Yaskawa INFORM job: driller_case_upwards_planes_program.JBI

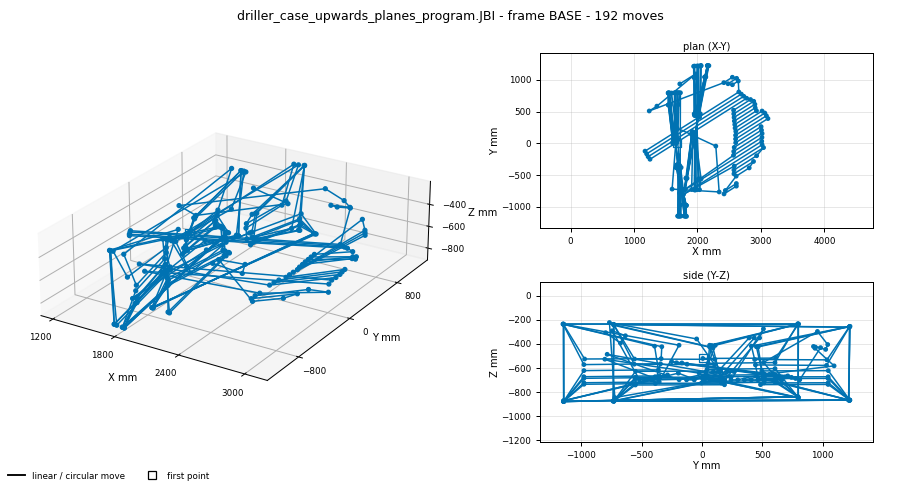
[picture p0: tool path of driller_case_upwards_planes_program.JBI in frame BASE, 192 of 196 moves have a stored position in this frame; points joined in program order, loops and branches not executed]
/JOB
//NAME driller_case_upwards_planes_program
//POS
///NPOS 192,0,192,0,0,0
///TOOL 0
///POSTYPE BASE
///RECTAN
///RCONF 0,0,0,0,0,0,0,0,0,0,0,0,0,0,0,0,0,0,0,0,0,0,0,0
C00000=1673.431880,7.470572,-520.659280,175.000000,-87.408482,-5.000000
C00001=1701.430434,612.195440,-517.792634,5.000000,-89.787348,-140.532242
C00002=1730.822135,797.239311,-237.810218,175.000000,-61.554488,-43.406673
C00003=1724.400104,-1148.148230,-235.635493,175.000000,-56.840650,28.530040
C00004=1729.963488,-971.443104,-525.203951,175.000000,-89.826502,-50.531598
C00005=1674.986268,-337.641847,-522.278767,168.678223,-90.000000,5.000000
C00006=1704.945690,-332.291816,-423.533285,5.000000,-42.547616,175.000000
C00007=1691.135780,-1145.204123,-238.489082,175.000000,-58.717311,26.416525
C00008=1739.409858,-1145.531949,-872.838304,-5.000000,-56.170316,-151.289669
C00009=1742.002509,-379.860852,-686.285449,175.000000,-48.174345,-17.109685
C00010=1678.244549,-343.199867,-564.964424,168.678223,-90.000000,5.000000
C00011=1818.384608,-977.621480,-571.536946,-175.000000,-89.631981,-46.846842
C00012=1826.808543,-1150.833072,-235.822537,175.000000,-54.888634,30.707899
C00013=1590.979545,793.251519,-233.985937,-175.000000,-62.535779,-40.616460
C00014=1571.245197,605.149655,-554.917240,5.000000,-89.484561,-136.850153
C00015=1625.513935,50.641867,-560.809912,168.678223,-90.000000,5.000000
C00016=1689.473871,63.888821,-411.282587,-5.000000,-48.045317,175.000000
C00017=1708.256775,799.356476,-235.389466,175.000000,-61.004563,-44.985899
C00018=1636.215691,796.253953,-843.502997,-5.000000,-63.369743,139.463298
C00019=1641.861992,13.097528,-670.904228,175.000000,-43.584726,-21.662339
C00020=1619.863907,43.091049,-610.639771,168.678223,-90.000000,5.000000
C00021=1564.744394,605.389718,-604.672433,5.000000,-89.485299,-136.858461
C00022=1558.133538,794.132963,-838.862886,5.000000,-63.890650,140.856457
C00023=1793.575292,-1145.031741,-876.264127,5.000000,-55.710812,-151.382699
C00024=1811.384412,-977.382379,-621.271160,175.000000,-89.632395,-46.855158
C00025=1673.763040,-360.368406,-614.890343,168.678223,-90.000000,5.000000
C00026=1713.133832,-392.278475,-418.917620,5.000000,-45.513699,161.896712
C00027=1701.888861,-1146.465321,-236.949035,175.000000,-57.847486,27.323797
C00028=1714.482776,-1144.136050,-870.078236,-5.000000,-56.959520,-152.294224
C00029=1719.658713,-351.013457,-679.536032,175.000000,-45.302626,-5.000000
C00030=1674.759987,-354.429105,-664.960497,168.678223,-90.000000,5.000000
C00031=1823.436094,-977.958927,-671.848021,175.000000,-89.610377,-46.409872
C00032=1809.321792,-1145.234620,-877.559004,5.000000,-55.428903,-151.169659
C00033=1544.248518,793.640543,-837.946269,5.000000,-64.024640,141.178755
C00034=1549.995593,604.768012,-654.123768,5.000000,-89.445413,-136.413643
C00035=1616.889276,32.814080,-660.602958,168.678223,-90.000000,5.000000
C00036=1669.829005,80.581913,-413.436350,5.000000,-46.334068,-175.000000
C00037=1682.622532,797.248951,-235.622802,175.000000,-61.552203,-43.413607
C00038=1656.620159,798.095359,-846.102626,5.000000,-62.596024,138.067586
C00039=1655.982659,0.583805,-677.340283,175.000000,-46.582826,-23.977786
C00040=1614.845882,21.413497,-710.613338,168.678223,-90.000000,5.000000
C00041=1544.922944,604.889358,-703.953307,5.000000,-89.440488,-136.359327
C00042=1541.265869,793.579835,-837.776448,5.000000,-64.040832,141.218191
C00043=1809.966137,-1145.258187,-877.659798,5.000000,-55.394158,-151.143981
C00044=1821.644860,-977.832954,-721.815313,175.000000,-89.607710,-46.355496
C00045=1671.662160,-353.900735,-714.869605,168.678223,-90.000000,5.000000
C00046=1694.918489,-189.479139,-411.049691,5.000000,-48.693566,-162.669170
C00047=1688.735226,-1145.992617,-237.083073,175.000000,-58.161087,26.984028
C00048=1714.386065,-1144.637206,-870.689055,5.000000,-56.663329,-151.932909
C00049=1723.789184,-403.538739,-698.708952,175.000000,-54.643933,-34.099882
C00050=1673.691517,-382.283167,-678.538009,168.678223,-90.000000,5.000000
C00051=1821.794903,-977.808560,-685.265560,175.000000,-89.602307,-46.245060
C00052=1812.732992,-1145.305389,-877.931109,5.000000,-55.323257,-151.091931
C00053=1536.659104,793.456173,-837.497478,-5.000000,-64.073595,141.298327
C00054=1538.402248,604.904947,-667.123556,-5.000000,-89.430451,-136.249014
C00055=1612.340142,12.697218,-673.988201,168.678223,-90.000000,5.000000
C00056=1668.454091,110.569857,-412.045848,5.000000,-46.959807,-174.665225
C00057=1681.902703,797.234172,-235.601339,-175.000000,-61.556609,-43.402511
C00058=1656.233440,798.109144,-846.096344,5.000000,-62.590789,138.057175
C00059=1656.170573,2.028916,-680.034745,-175.000000,-47.980448,-27.377056
C00060=1610.322073,-2.559617,-724.017037,168.678223,-90.000000,5.000000
C00061=1545.419504,606.009907,-717.420022,-5.000000,-89.472373,-136.713354
C00062=1547.396406,793.973294,-838.282370,-5.000000,-63.934611,140.961437
C00063=1792.490907,-1145.099774,-876.404413,5.000000,-55.619211,-151.312650
C00064=1800.788436,-976.746038,-734.385420,175.000000,-89.625178,-46.709903
C00065=1663.430936,-385.311442,-728.138889,180.000000,-60.000000,0.000000
C00066=2418.072893,-797.339000,-307.192250,175.000000,-13.138131,5.000000
C00067=2612.434723,-674.639778,-393.619264,175.000000,-13.138131,5.000000
C00068=2612.338702,-633.486964,-332.637264,175.000000,-13.138131,5.000000
C00069=2439.090274,-742.857448,-291.122264,175.000000,-13.138131,5.000000
C00070=2609.232584,-517.188349,-698.109264,175.000000,-13.138131,5.000000
C00071=2815.107824,-387.220793,-671.983264,175.000000,-13.138131,5.000000
C00072=2882.831238,-285.337748,-656.650264,175.000000,-13.138131,5.000000
C00073=2574.452592,-480.014964,-698.349264,175.000000,-13.138131,5.000000
C00074=2574.249107,-421.013680,-696.275264,175.000000,-13.138131,5.000000
C00075=2931.745166,-195.328994,-642.567264,175.000000,-13.138131,5.000000
C00076=3040.631451,-67.460124,-690.751264,175.000000,-13.138131,5.000000
C00077=2579.605431,-358.502529,-697.708264,175.000000,-13.138131,5.000000
C00078=1780.417411,-803.894423,-526.918264,175.000000,-13.138131,5.000000
C00079=3018.335870,-22.405421,-642.237264,175.000000,-13.138131,5.000000
C00080=3012.500702,33.040622,-630.532264,175.000000,-13.138131,5.000000
C00081=1716.986018,-784.808462,-486.219264,175.000000,-13.138131,5.000000
C00082=2567.445798,-188.789589,-697.222264,175.000000,-13.138131,5.000000
C00083=3015.932444,94.336798,-631.217264,175.000000,-13.138131,5.000000
C00084=3018.491529,155.082073,-626.978264,175.000000,-13.138131,5.000000
C00085=2571.014527,-127.406933,-697.829264,175.000000,-13.138131,5.000000
C00086=2578.759665,-63.387741,-698.559264,175.000000,-13.138131,5.000000
C00087=3008.587342,207.959374,-627.283264,175.000000,-13.138131,5.000000
C00088=3002.687909,263.364847,-628.708264,175.000000,-13.138131,5.000000
C00089=2601.758547,10.261031,-697.750264,175.000000,-13.138131,5.000000
C00090=2600.088796,68.336671,-698.106264,175.000000,-13.138131,5.000000
C00091=3110.624587,390.634237,-350.634264,175.000000,-13.138131,5.000000
C00092=3086.098318,434.280723,-350.923264,175.000000,-13.138131,5.000000
C00093=2600.297118,127.597926,-698.488264,175.000000,-13.138131,5.000000
C00094=2603.303524,188.625591,-697.822264,175.000000,-13.138131,5.000000
C00095=3061.064690,477.606917,-350.373264,175.000000,-13.138131,5.000000
C00096=3017.690039,509.354554,-275.549264,175.000000,-13.138131,5.000000
C00097=2592.388002,240.864444,-698.256264,175.000000,-13.138131,5.000000
C00098=2587.301189,296.782918,-697.884264,175.000000,-13.138131,5.000000
C00099=2929.507142,512.815070,-646.336264,175.000000,-13.138131,5.000000
C00100=2909.851518,559.536359,-652.328264,175.000000,-13.138131,5.000000
C00101=2580.862263,351.847814,-698.019264,175.000000,-13.138131,5.000000
C00102=2576.339464,408.122346,-698.387264,175.000000,-13.138131,5.000000
C00103=2904.740182,615.439352,-696.121264,175.000000,-13.138131,5.000000
C00104=2886.403691,662.993401,-697.340264,175.000000,-13.138131,5.000000
C00105=2571.376107,464.118757,-698.288264,175.000000,-13.138131,5.000000
C00106=2568.806639,521.626413,-697.221264,175.000000,-13.138131,5.000000
C00107=2835.976752,690.288980,-673.466264,175.000000,-13.138131,5.000000
C00108=2774.286445,710.474076,-664.905264,175.000000,-13.138131,5.000000
C00109=1251.445386,-250.884509,-547.070264,175.000000,-13.138131,5.000000
C00110=1222.182922,-210.227949,-556.282264,175.000000,-13.138131,5.000000
C00111=2729.668764,741.436999,-677.026264,175.000000,-13.138131,5.000000
C00112=2690.657399,775.939148,-686.387264,175.000000,-13.138131,5.000000
C00113=1198.557215,-166.012945,-557.802264,175.000000,-13.138131,5.000000
C00114=1173.125310,-122.938180,-568.494264,175.000000,-13.138131,5.000000
C00115=2651.104851,810.099652,-696.529264,175.000000,-13.138131,5.000000
C00116=2643.398138,982.623688,-430.995264,175.000000,-13.138131,5.000000
C00117=2550.399255,923.914164,-421.281264,175.000000,-13.138131,5.000000
C00118=2481.149301,939.326909,-426.588264,175.000000,-13.138131,5.000000
C00119=2616.445002,1024.738110,-445.606264,175.000000,-13.138131,5.000000
C00120=2549.748754,1041.762992,-405.392264,175.000000,-13.138131,5.000000
C00121=2414.820888,956.584003,-297.084264,175.000000,-13.138131,5.000000
C00122=1239.226227,510.088279,-553.661264,175.000000,-13.138131,5.000000
C00123=1360.051207,586.364219,-645.180264,175.000000,-13.138131,5.000000
C00124=1971.096569,1094.552710,-581.948264,175.000000,-13.138131,5.000000
C00125=1720.950038,936.637008,-436.438264,175.000000,-13.138131,5.000000
C00126=1961.484996,107.194191,-528.136914,5.000000,-87.762077,175.000000
C00127=2016.650761,-558.205833,-525.321042,5.000000,-89.841698,129.060213
C00128=1989.641452,-729.842232,-241.045760,175.000000,-57.590997,26.248990
C00129=1997.453896,1220.092504,-260.476656,-175.000000,-62.729371,-42.375589
C00130=1987.427131,1034.868670,-532.157780,175.000000,-89.803316,39.059669
C00131=1960.156670,436.797064,-529.555779,167.889080,-90.000000,5.000000
C00132=2032.382048,409.596982,-418.437173,-5.000000,-51.077351,163.119403
C00133=2054.997730,1226.570891,-254.753398,175.000000,-61.067124,-47.210966
C00134=1939.009741,1213.927494,-864.805716,5.000000,-64.011021,140.374043
C00135=1947.622597,464.514384,-680.611039,175.000000,-39.536143,-5.000000
C00136=1952.014832,443.273018,-574.460068,167.889080,-90.000000,5.000000
C00137=1948.276945,1032.014046,-578.095382,175.000000,-89.712556,40.386055
C00138=1952.492216,1218.817292,-263.193512,175.000000,-63.172057,-41.437844
C00139=2031.818883,-730.783852,-237.814917,175.000000,-56.842528,26.968983
C00140=2056.236526,-560.610843,-568.391185,5.000000,-89.779417,130.387161
C00141=1969.048653,105.201390,-572.392321,167.889080,-90.000000,5.000000
C00142=2288.843492,-43.671885,-359.161426,5.000000,-71.416390,160.782079
C00143=2341.409332,-766.085094,-223.316094,175.000000,-55.190941,48.507226
C00144=1599.653871,-721.210506,-844.569748,-5.000000,-74.132634,-161.793602
C00145=1676.842950,239.149767,-675.094607,-163.063119,-22.671233,-6.694605
C00146=1907.112237,138.286849,-624.988576,167.889080,-90.000000,5.000000
C00147=1816.394484,-549.757259,-627.429473,-175.000000,-89.858176,-56.659513
C00148=1791.168636,-728.786980,-873.539578,-5.000000,-59.243967,-155.889318
C00149=2179.400692,1224.243522,-865.643847,5.000000,-59.867382,132.065978
C00150=2131.014554,1046.554867,-621.689313,5.000000,-89.855924,-146.659870
C00151=1977.994382,495.990739,-623.702030,167.889080,-90.000000,5.000000
C00152=2039.534805,451.255661,-423.680556,5.000000,-48.510324,160.054868
C00153=2051.362128,1223.186154,-256.283333,175.000000,-61.751329,-44.707154
C00154=2007.613275,1216.620546,-865.296779,5.000000,-62.727347,138.304036
C00155=2005.199291,513.306929,-683.985357,175.000000,-42.825788,-5.000000
C00156=1974.556380,504.642963,-673.910864,167.889080,-90.000000,5.000000
C00157=2117.406414,1045.523171,-672.227168,5.000000,-89.876178,-146.282104
C00158=2162.728234,1223.977001,-865.957873,5.000000,-60.006590,132.329966
C00159=1800.141078,-729.234842,-873.540455,5.000000,-59.094919,-155.630777
C00160=1826.073230,-550.510492,-677.113133,175.000000,-89.879710,-56.281844
C00161=1909.425615,151.613602,-674.992035,167.889080,-90.000000,5.000000
C00162=1926.980134,91.571093,-433.363326,5.000000,-45.138585,154.790994
C00163=1907.398248,-728.573806,-246.303114,175.000000,-58.547302,25.326984
C00164=1966.396538,-735.978282,-874.194316,-5.000000,-56.003080,-151.232974
C00165=1964.617837,164.094456,-692.828761,175.000000,-47.689988,-5.000000
C00166=1914.152160,162.220658,-724.889909,167.889080,-90.000000,5.000000
C00167=1823.958368,-550.457109,-727.222082,175.000000,-89.869493,-56.461613
C00168=1795.480622,-729.022635,-873.554636,-5.000000,-59.166165,-155.753634
C00169=2170.258774,1224.104798,-865.823608,5.000000,-59.940629,132.204194
C00170=2126.360175,1045.707967,-721.930144,5.000000,-89.866501,-146.461917
C00171=1981.075805,512.627954,-723.727799,167.889080,-90.000000,5.000000
C00172=2044.166999,465.174961,-425.385194,-5.000000,-47.585730,162.061091
C00173=2055.148595,1222.784222,-256.359125,175.000000,-61.858152,-44.406299
C00174=2020.313082,1216.978526,-865.158762,5.000000,-62.582587,138.030421
C00175=2017.125609,510.220351,-683.994633,175.000000,-43.115600,-5.293268
C00176=1978.339507,518.918494,-687.296876,167.889080,-90.000000,5.000000
C00177=2114.133291,1044.672008,-685.810947,5.000000,-89.887063,-146.081316
C00178=2154.956327,1223.831881,-866.084078,5.000000,-60.079673,132.470975
C00179=1805.952083,-729.469729,-873.502157,-5.000000,-59.014758,-155.494032
C00180=1835.127568,-551.217347,-690.244850,175.000000,-89.891051,-56.081102
C00181=1916.971035,172.700277,-688.259266,167.889080,-90.000000,5.000000
C00182=1963.683735,63.570575,-424.933376,5.000000,-48.631320,153.774363
C00183=1952.299153,-730.683848,-241.301563,175.000000,-57.021308,26.858770
C00184=1950.745317,-733.584538,-871.676569,5.000000,-57.371083,-152.947455
C00185=1956.699130,164.411626,-689.093377,-175.000000,-45.459043,5.000000
C00186=1916.855659,186.914842,-738.361322,167.889080,-90.000000,5.000000
C00187=1828.776803,-551.231476,-740.522460,175.000000,-89.883579,-56.213515
C00188=1797.211740,-729.314958,-873.718800,5.000000,-59.067811,-155.584247
C00189=2155.172709,1223.927878,-866.192704,5.000000,-60.031479,132.377870
C00190=2115.910105,1044.752779,-735.790520,-5.000000,-89.879874,-146.213759
C00191=1971.166504,485.284250,-737.476298,180.000000,-60.000000,0.000000
///POSTYPE PULSE
///PULSE
EC00000=173056.0
EC00001=173056.0
EC00002=173056.0
EC00003=173056.0
EC00004=173056.0
EC00005=173056.0
EC00006=173056.0
EC00007=173056.0
EC00008=173056.0
EC00009=173056.0
EC00010=173056.0
EC00011=173056.0
EC00012=173056.0
EC00013=173056.0
EC00014=173056.0
EC00015=173056.0
EC00016=173056.0
EC00017=173056.0
EC00018=173056.0
EC00019=173056.0
EC00020=173056.0
EC00021=173056.0
EC00022=173056.0
EC00023=173056.0
EC00024=173056.0
EC00025=173056.0
EC00026=173056.0
EC00027=173056.0
EC00028=173056.0
EC00029=173056.0
EC00030=173056.0
EC00031=173056.0
EC00032=173056.0
EC00033=173056.0
EC00034=173056.0
EC00035=173056.0
EC00036=173056.0
EC00037=173056.0
EC00038=173056.0
EC00039=173056.0
EC00040=173056.0
EC00041=173056.0
EC00042=173056.0
EC00043=173056.0
EC00044=173056.0
EC00045=173056.0
EC00046=173056.0
EC00047=173056.0
EC00048=173056.0
EC00049=173056.0
EC00050=173056.0
EC00051=173056.0
EC00052=173056.0
EC00053=173056.0
EC00054=173056.0
EC00055=173056.0
EC00056=173056.0
EC00057=173056.0
EC00058=173056.0
EC00059=173056.0
EC00060=173056.0
EC00061=173056.0
EC00062=173056.0
EC00063=173056.0
EC00064=173056.0
EC00065=173056.0
EC00066=309248.0
EC00067=309248.0
EC00068=309248.0
EC00069=309248.0
EC00070=309248.0
EC00071=309248.0
EC00072=309248.0
EC00073=309248.0
EC00074=309248.0
EC00075=309248.0
EC00076=309248.0
EC00077=309248.0
EC00078=309248.0
EC00079=309248.0
EC00080=309248.0
EC00081=309248.0
EC00082=309248.0
EC00083=309248.0
EC00084=309248.0
EC00085=309248.0
EC00086=309248.0
EC00087=309248.0
EC00088=309248.0
EC00089=309248.0
EC00090=309248.0
EC00091=309248.0
EC00092=309248.0
EC00093=309248.0
EC00094=309248.0
EC00095=309248.0
EC00096=309248.0
EC00097=309248.0
EC00098=309248.0
EC00099=309248.0
EC00100=309248.0
EC00101=309248.0
EC00102=309248.0
EC00103=309248.0
EC00104=309248.0
EC00105=309248.0
EC00106=309248.0
EC00107=309248.0
EC00108=309248.0
EC00109=309248.0
EC00110=309248.0
EC00111=309248.0
EC00112=309248.0
EC00113=309248.0
EC00114=309248.0
EC00115=309248.0
EC00116=309248.0
EC00117=309248.0
EC00118=309248.0
EC00119=309248.0
EC00120=309248.0
EC00121=309248.0
EC00122=309248.0
EC00123=309248.0
EC00124=309248.0
EC00125=309248.0
EC00126=356352.0
EC00127=356352.0
EC00128=356352.0
EC00129=356352.0
EC00130=356352.0
EC00131=356352.0
EC00132=356352.0
EC00133=356352.0
EC00134=356352.0
EC00135=356352.0
EC00136=356352.0
EC00137=356352.0
EC00138=356352.0
EC00139=356352.0
EC00140=356352.0
EC00141=356352.0
EC00142=356352.0
EC00143=356352.0
EC00144=356352.0
EC00145=356352.0
EC00146=356352.0
EC00147=356352.0
EC00148=356352.0
EC00149=356352.0
EC00150=356352.0
EC00151=356352.0
EC00152=356352.0
EC00153=356352.0
EC00154=356352.0
EC00155=356352.0
EC00156=356352.0
EC00157=356352.0
EC00158=356352.0
EC00159=356352.0
EC00160=356352.0
EC00161=356352.0
EC00162=356352.0
EC00163=356352.0
EC00164=356352.0
EC00165=356352.0
EC00166=356352.0
EC00167=356352.0
EC00168=356352.0
EC00169=356352.0
EC00170=356352.0
EC00171=356352.0
EC00172=356352.0
EC00173=356352.0
EC00174=356352.0
EC00175=356352.0
EC00176=356352.0
EC00177=356352.0
EC00178=356352.0
EC00179=356352.0
EC00180=356352.0
EC00181=356352.0
EC00182=356352.0
EC00183=356352.0
EC00184=356352.0
EC00185=356352.0
EC00186=356352.0
EC00187=356352.0
EC00188=356352.0
EC00189=356352.0
EC00190=356352.0
EC00191=356352.0
//INST
///DATE 2023/08/04 15:15
///ATTR SC,RW,RJ
////FRAME BASE
///GROUP1 RB1,ST1
NOP
MOVJ P009 EX000 VJ=15.00
MOVJ C00000 EC00000 VJ=15.0
CALL JOB:SPYON
MOVL C00001 EC00001 V=150.0
MOVL C00002 EC00002 V=150.0
MOVL C00003 EC00003 V=150.0
MOVL C00004 EC00004 V=150.0
MOVL C00005 EC00005 V=150.0
MOVL C00006 EC00006 V=150.0
MOVL C00007 EC00007 V=150.0
MOVL C00008 EC00008 V=150.0
MOVL C00009 EC00009 V=150.0
MOVL C00010 EC00010 V=150.0
MOVL C00011 EC00011 V=150.0
MOVL C00012 EC00012 V=150.0
MOVL C00013 EC00013 V=150.0
MOVL C00014 EC00014 V=150.0
MOVL C00015 EC00015 V=150.0
MOVL C00016 EC00016 V=150.0
MOVL C00017 EC00017 V=150.0
MOVL C00018 EC00018 V=150.0
MOVL C00019 EC00019 V=150.0
MOVL C00020 EC00020 V=150.0
MOVL C00021 EC00021 V=150.0
MOVL C00022 EC00022 V=150.0
MOVL C00023 EC00023 V=150.0
MOVL C00024 EC00024 V=150.0
MOVL C00025 EC00025 V=150.0
MOVL C00026 EC00026 V=150.0
MOVL C00027 EC00027 V=150.0
MOVL C00028 EC00028 V=150.0
MOVL C00029 EC00029 V=150.0
MOVL C00030 EC00030 V=150.0
MOVL C00031 EC00031 V=150.0
MOVL C00032 EC00032 V=150.0
MOVL C00033 EC00033 V=150.0
MOVL C00034 EC00034 V=150.0
MOVL C00035 EC00035 V=150.0
MOVL C00036 EC00036 V=150.0
MOVL C00037 EC00037 V=150.0
MOVL C00038 EC00038 V=150.0
MOVL C00039 EC00039 V=150.0
MOVL C00040 EC00040 V=150.0
MOVL C00041 EC00041 V=150.0
MOVL C00042 EC00042 V=150.0
MOVL C00043 EC00043 V=150.0
MOVL C00044 EC00044 V=150.0
MOVL C00045 EC00045 V=150.0
MOVL C00046 EC00046 V=150.0
MOVL C00047 EC00047 V=150.0
MOVL C00048 EC00048 V=150.0
MOVL C00049 EC00049 V=150.0
MOVL C00050 EC00050 V=150.0
MOVL C00051 EC00051 V=150.0
MOVL C00052 EC00052 V=150.0
MOVL C00053 EC00053 V=150.0
MOVL C00054 EC00054 V=150.0
MOVL C00055 EC00055 V=150.0
MOVL C00056 EC00056 V=150.0
MOVL C00057 EC00057 V=150.0
MOVL C00058 EC00058 V=150.0
MOVL C00059 EC00059 V=150.0
MOVL C00060 EC00060 V=150.0
MOVL C00061 EC00061 V=150.0
MOVL C00062 EC00062 V=150.0
MOVL C00063 EC00063 V=150.0
MOVL C00064 EC00064 V=150.0
MOVL C00065 EC00065 V=150.0
CALL JOB:SPYOF
MOVJ P009 VJ=15.00
MOVJ C00066 EC00066 VJ=15.0
CALL JOB:SPYON
MOVL C00067 EC00067 V=150.0
MOVL C00068 EC00068 V=150.0
MOVL C00069 EC00069 V=150.0
MOVL C00070 EC00070 V=150.0
MOVL C00071 EC00071 V=150.0
MOVL C00072 EC00072 V=150.0
MOVL C00073 EC00073 V=150.0
MOVL C00074 EC00074 V=150.0
MOVL C00075 EC00075 V=150.0
MOVL C00076 EC00076 V=150.0
MOVL C00077 EC00077 V=150.0
MOVL C00078 EC00078 V=150.0
MOVL C00079 EC00079 V=150.0
MOVL C00080 EC00080 V=150.0
MOVL C00081 EC00081 V=150.0
MOVL C00082 EC00082 V=150.0
MOVL C00083 EC00083 V=150.0
MOVL C00084 EC00084 V=150.0
MOVL C00085 EC00085 V=150.0
MOVL C00086 EC00086 V=150.0
MOVL C00087 EC00087 V=150.0
MOVL C00088 EC00088 V=150.0
MOVL C00089 EC00089 V=150.0
MOVL C00090 EC00090 V=150.0
MOVL C00091 EC00091 V=150.0
MOVL C00092 EC00092 V=150.0
MOVL C00093 EC00093 V=150.0
MOVL C00094 EC00094 V=150.0
MOVL C00095 EC00095 V=150.0
MOVL C00096 EC00096 V=150.0
MOVL C00097 EC00097 V=150.0
MOVL C00098 EC00098 V=150.0
MOVL C00099 EC00099 V=150.0
MOVL C00100 EC00100 V=150.0
MOVL C00101 EC00101 V=150.0
MOVL C00102 EC00102 V=150.0
MOVL C00103 EC00103 V=150.0
MOVL C00104 EC00104 V=150.0
MOVL C00105 EC00105 V=150.0
MOVL C00106 EC00106 V=150.0
MOVL C00107 EC00107 V=150.0
MOVL C00108 EC00108 V=150.0
MOVL C00109 EC00109 V=150.0
MOVL C00110 EC00110 V=150.0
MOVL C00111 EC00111 V=150.0
MOVL C00112 EC00112 V=150.0
MOVL C00113 EC00113 V=150.0
MOVL C00114 EC00114 V=150.0
MOVL C00115 EC00115 V=150.0
MOVL C00116 EC00116 V=150.0
MOVL C00117 EC00117 V=150.0
MOVL C00118 EC00118 V=150.0
MOVL C00119 EC00119 V=150.0
MOVL C00120 EC00120 V=150.0
MOVL C00121 EC00121 V=150.0
MOVL C00122 EC00122 V=150.0
MOVL C00123 EC00123 V=150.0
MOVL C00124 EC00124 V=150.0
MOVL C00125 EC00125 V=150.0
CALL JOB:SPYOF
MOVJ P009 VJ=15.00
MOVJ C00126 EC00126 VJ=15.0
CALL JOB:SPYON
MOVL C00127 EC00127 V=150.0
MOVL C00128 EC00128 V=150.0
MOVL C00129 EC00129 V=150.0
MOVL C00130 EC00130 V=150.0
MOVL C00131 EC00131 V=150.0
MOVL C00132 EC00132 V=150.0
MOVL C00133 EC00133 V=150.0
MOVL C00134 EC00134 V=150.0
MOVL C00135 EC00135 V=150.0
MOVL C00136 EC00136 V=150.0
MOVL C00137 EC00137 V=150.0
MOVL C00138 EC00138 V=150.0
MOVL C00139 EC00139 V=150.0
MOVL C00140 EC00140 V=150.0
MOVL C00141 EC00141 V=150.0
MOVL C00142 EC00142 V=150.0
MOVL C00143 EC00143 V=150.0
MOVL C00144 EC00144 V=150.0
MOVL C00145 EC00145 V=150.0
MOVL C00146 EC00146 V=150.0
MOVL C00147 EC00147 V=150.0
MOVL C00148 EC00148 V=150.0
MOVL C00149 EC00149 V=150.0
MOVL C00150 EC00150 V=150.0
MOVL C00151 EC00151 V=150.0
MOVL C00152 EC00152 V=150.0
MOVL C00153 EC00153 V=150.0
MOVL C00154 EC00154 V=150.0
MOVL C00155 EC00155 V=150.0
MOVL C00156 EC00156 V=150.0
MOVL C00157 EC00157 V=150.0
MOVL C00158 EC00158 V=150.0
MOVL C00159 EC00159 V=150.0
MOVL C00160 EC00160 V=150.0
MOVL C00161 EC00161 V=150.0
MOVL C00162 EC00162 V=150.0
MOVL C00163 EC00163 V=150.0
MOVL C00164 EC00164 V=150.0
MOVL C00165 EC00165 V=150.0
MOVL C00166 EC00166 V=150.0
MOVL C00167 EC00167 V=150.0
MOVL C00168 EC00168 V=150.0
MOVL C00169 EC00169 V=150.0
MOVL C00170 EC00170 V=150.0
MOVL C00171 EC00171 V=150.0
MOVL C00172 EC00172 V=150.0
MOVL C00173 EC00173 V=150.0
MOVL C00174 EC00174 V=150.0
MOVL C00175 EC00175 V=150.0
MOVL C00176 EC00176 V=150.0
MOVL C00177 EC00177 V=150.0
MOVL C00178 EC00178 V=150.0
MOVL C00179 EC00179 V=150.0
MOVL C00180 EC00180 V=150.0
MOVL C00181 EC00181 V=150.0
MOVL C00182 EC00182 V=150.0
MOVL C00183 EC00183 V=150.0
MOVL C00184 EC00184 V=150.0
MOVL C00185 EC00185 V=150.0
MOVL C00186 EC00186 V=150.0
MOVL C00187 EC00187 V=150.0
MOVL C00188 EC00188 V=150.0
MOVL C00189 EC00189 V=150.0
MOVL C00190 EC00190 V=150.0
MOVL C00191 EC00191 V=150.0
CALL JOB:SPYOF
MOVJ P009 VJ=15.00
END
